// TIA Portal V18 export
DATA_BLOCK "Re-filling Sequence DB"   // DB103
{ S7_Optimized_Access := 'TRUE' }
VERSION : 0.1
// stored: AutoNumber true, DBAccessibleFromOPCUA true, IsOnlyStoredInLoadMemory false, IsRetainMemResEnabled false, IsWriteProtectedInAS false, MemoryReserve 100
   VAR
      "Refilling Enable" : Bool;
      "Refilling manual Comp A" : Bool;
      "Refilling manual Comp B" : Bool;
      "Refiling ValveA ON" : Bool;
      "Refiling ValveA ON Manual" : Bool;
      "Refilling Manual Componet A" : Bool;
      "Refilling Manual Componet B" : Bool;
      "Refiling ValveB ON" : Bool;
      "Refiling ValveB ON Manual" : Bool;
      "AODD Pump Component A ON" : Bool;
      "AODD Pump Component A ON- Manual" : Bool;
      "AODD Pump Component B ON" : Bool;
      "AODD Pump Component B ON- Manual" : Bool;
   END_VAR
   VAR RETAIN
      "AODD  componet A  ON delay" : Time;
      "AODD  componet B  ON delay" : Time;
   END_VAR
   VAR
      "Compare Re-fillingFilling sequence A" : Struct
         "Start Compare" : Bool;
         "Re-filling % in 30 Sec" : Real;
         "Excpected Level" : Real;
         "Refilling Error" : Bool;
      END_STRUCT;
      "Compare Filling sequence b" : Struct
         "Start Compare" : Bool;
         "Re-filling % in 30 Sec" : Real;
         "Excpected Level" : Real;
         "Refilling Error" : Bool;
      END_STRUCT;
   END_VAR
   VAR RETAIN
      "A valve off pump off delay" : DInt;
      "B valve off pump off delay" : DInt;
   END_VAR
   VAR
      temp1 : Bool;
      temp2 : Bool;
   END_VAR
BEGIN
END_DATA_BLOCK
